Fanuc KAREL source: NC0064.KL

-- PROVISIONAL review KL for V940-1; original PC SHA256 55095405fa6989c3c1444c9833b5bc0aed306e42b3fe563aace35c466cfc4728
-- Incomplete behavior may be omitted. Consult companion uncertainty JSON. Do not deploy.
PROGRAM NC0064
%NOLOCKGROUP
-- UNRESOLVED_LOCAL_POOL 4 cells at code offset 3; source declarations unknown
-- DIRECT_LOCAL_WORD_ACCESS alone does not prove INTEGER, REAL, or BOOLEAN
BEGIN
  -- V9_EXPOSED_INDEXED_TABLE_HINT layout=0001; 6 counted words exposed once; source arms/runtime held
  -- V9_FOOTER_20_HINT 3 numerical footer links; VM transfer unproved
  -- UNRESOLVED_PC offsets 0-8; opcodes 2B,2C,7B
  -- UNRESOLVED_PC offsets 13-20; opcodes 9D,23
  -- UNRESOLVED_PC offsets 25-54; opcodes 9D,23,9E,2E,22,7A
  -- UNRESOLVED_PC offsets 59-88; opcodes 9D,23,9E,2E,22,7A
  -- UNRESOLVED_PC offsets 93-122; opcodes 9D,23,9E,2E,22,7A
  -- UNRESOLVED_PC offsets 127-141; opcodes 21,9D,52,23
  -- UNRESOLVED_PC offsets 146-161; opcodes 20,2C,23
  -- UNRESOLVED_PC offsets 166-181; opcodes 20,2C,23
  -- UNRESOLVED_PC offsets 186-201; opcodes 20,2C,23
  -- UNRESOLVED_PC offsets 206-210; opcodes 7F
  -- UNRESOLVED_PC offsets 215-219; opcodes 27,AA
  -- UNRESOLVED_PC offsets 224-228; opcodes 7F
END NC0064
